//==================================================================================================
//								RJM Maszyny sp. z o.o.
//									22.06.2022
//	Obsługa przycisku ze stykiem NO
// 	v1.0	|| TC v 3.1.4024.22		|| - pierwsza wersja
//==================================================================================================
FUNCTION_BLOCK FB_Przycisk_NO IMPLEMENTS ITF_Przycisk
VAR
	bStyk							AT %I*	: BOOL;
	bPodswietlenie					AT %Q*	: BOOL;
END_VAR

PROPERTY CzyNacisniety : BOOL
GET
CzyNacisniety								:= bStyk;
END_GET
END_PROPERTY

PROPERTY Podswietlenie : BOOL
SET
bPodswietlenie								:= Podswietlenie;
END_SET
END_PROPERTY

END_FUNCTION_BLOCK

(* stored: Version 1.1.0.1, ProductVersion 3.1.4024.11
   POU FB_Przycisk_NO: Id {3ba1b16e-e023-47d3-b391-378d8339a797}, SpecialFunc None
   Property CzyNacisniety: Id {89bb073c-3b68-48b5-9fc4-2ca0e7c833a4}
   Get Get: Id {9c183c44-60d7-4cc2-ba81-9e7a9b76996f}
   Property Podswietlenie: Id {6693ee11-fedc-4f68-b760-80b9eb65c982}
   Set Set: Id {c8d194b1-47e5-40e4-9ea6-86728638cc25} *)
